FUNCTION_BLOCK Gen
  (* Standard: 61499-2 *)
  (* Version 0.1, 2017-00-01, hpea485, UOA *)
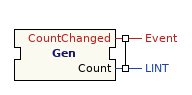
  EVENT_OUTPUT
    CountChanged WITH Count;
  END_EVENT
  VAR_OUTPUT
    Count : LINT := 0;
  END_VAR
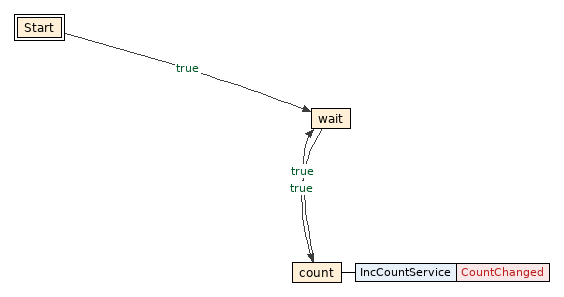
  EC_STATES
    Start;
    count : IncCountService -> CountChanged;
    wait;
  END_STATES
  EC_TRANSITIONS
    Start TO wait := true;
    count TO wait := true;
    wait TO count := true;
  END_TRANSITIONS
  ALGORITHM IncCountService IN C:
me->Count++;
  END_ALGORITHM
END_FUNCTION_BLOCK
